TYPE ST_StartupSafetyConfig :
STRUCT
    tEnableTimeout : TIME;
END_STRUCT
END_TYPE

(* stored: Version 1.1.0.1, ProductVersion 3.1.4026.20
   DUT ST_StartupSafetyConfig: Id {e7616d8b-b062-48c1-af49-a4f44b844829} *)
